# EPICS IOC start-up script: iocsh/ethercatmcAuxBitAsBiRecord.iocsh
ethercatmcCreateAsynParam $(MOTOR_PORT) $(AUX_BIT_NAME_P) Int32

dbLoadRecords("ethercatmcAuxBitAsBiRecord.template", "PREFIX=$(PREFIX), MOTOR_NAME=$(MOTOR_NAME), MOTOR_PORT=$(MOTOR_PORT), AXIS_NO=$(AXIS_NO), AUX_BIT_NAME_R=$(AUX_BIT_NAME_R), AUX_BIT_NAME_P=$(AUX_BIT_NAME_P)")
